{attribute addProperty BoxType "ELM2644-0000-0016"}
{attribute addProperty Id "Outputs_Channel_4AT %Q*Outputs_Channel_E6FE5E20162"}
{attribute addProperty CRC "1229103389"}
{attribute addProperty SizeInBites "16"}
{attribute addProperty SizeInBytes "2"}
TYPE DO_Group_4_Outputs_4942A11D :
STRUCT
	{attribute addProperty Name "Outputs_Channel_4"}
	Outputs_Channel_4 AT %Q* : Outputs_Channel_E6FE5E20;
END_STRUCT
END_TYPE

(* stored: Version 1.2.0.0, ProductVersion 3.1.4024.9
   DUT DO_Group_4_Outputs_4942A11D: Id {0372c687-a01b-4036-945a-13a10c480c09} *)
